// TIA Portal V20 export
TYPE "LKinCtrl_typeRetProfileDist"
   STRUCT
      dist : LReal;
      functionResult : DInt;
   END_STRUCT;
END_TYPE
